// TwinCAT 3 PLC project Database_Code
// ProgramVersion: 3.1.4026.16
// libraries:
//   Tc2_Standard, * (Beckhoff Automation GmbH)
//   Tc2_System, * (Beckhoff Automation GmbH)
//   Tc2_Utilities, * (Beckhoff Automation GmbH)
//   Tc3_Database, * (Beckhoff Automation GmbH)
// project tree:
//   DUTs/ ST_SensorData.TcDUT
//   GVLs/ Global_Variables.TcGVL
//   / PlcTask.TcTTO
//   POUs/ CapacitiveConvert.TcPOU, FB_BufferManager.TcPOU, EncoderConvert.TcPOU, FC_SQL_InsertCommands_Capacitief.TcPOU, FC_SQL_InsertCommands_Encoder.TcPOU, FC_SQL_InsertCommands_TempSensor.TcPOU, FC_SQL_InsertCommands_LoadCell.TcPOU, LoadcellConvert.TcPOU, MAIN.TcPOU, TempConvert.TcPOU, TestCase.TcPOU
// real-time tasks:
//   TASK PlcTask: cycle T#5ms, priority 20, ADS port 350
// I/O:
//   DEVICE Device 3 (EtherCAT), AmsNetId 10.100.5.10.4.1
//     Term 6 (EK1100) [EK1100 EtherCAT Coupler (2A E-Bus)]
//       Term 7 (EL3074) [EL3074 4Ch. Ana. Input +/-10V, +/-20mA]
//       Term 8 (EL5032) [EL5032 2Ch. EnDat Encoder]
//       Term 9 (EL3204) [EL3204 4Ch. Ana. Input PT100 (RTD)]
//       Term 10 (EL7031) [EL7031 1Ch. Stepper motor output stage (24V, 1.5A)]
//       Term 12 (EL1819) [EL1819 16Ch. Dig. Input 24V, 10µs]
//       Term 13 (EL4004) [EL4004 4Ch. Ana. Output 0-10V, 12bit]
//       Term 16 (EL2809) [EL2809 16Ch. Dig. Output 24V, 0.5A]
//       Term 17 (EL9011) [EL9011 End Terminal]
// variable links:
//   Database_Code/Database_Code Instance <-> Device 3 (EtherCAT)/Term 6 (EK1100)/Term 10 (EL7031)
//     PlcTask Inputs/MAIN.RealMotorPosition <-> ENC Status/Counter value
//     PlcTask Inputs/MAIN.iLichtSluisValue1 <-> STM Status/Status/Digital input 1
//     PlcTask Inputs/MAIN.iLichtSluisValue2 <-> STM Status/Status/Digital input 2
//     PlcTask Inputs/MAIN.iMotorBusy <-> POS Status/Status/Busy
//     PlcTask Inputs/MAIN.iMotorCalibrated <-> POS Status/Status/Calibrated
//     PlcTask Inputs/MAIN.iMotorReady <-> POS Status/Status/Ready to execute
//     PlcTask Inputs/MAIN.iMotorStatus <-> POS Status/Status/Error
//     PlcTask Inputs/MAIN.iMotorWarning <-> POS Status/Status/Warning
//     PlcTask Outputs/MAIN.oEnableStart <-> ENC Control/Control/Set counter
//     PlcTask Outputs/MAIN.oMotorEnable <-> STM Control/Control/Enable
//     PlcTask Outputs/MAIN.oMotorExecute <-> POS Control/Control/Execute
//     PlcTask Outputs/MAIN.oMotorPosition <-> POS Control/Target position
//     PlcTask Outputs/MAIN.oMotorReset <-> STM Control/Control/Reset
//     PlcTask Outputs/MAIN.oMotorStartType <-> POS Control/Start type
//     PlcTask Outputs/MAIN.oMotorVelocity <-> POS Control/Velocity
//     PlcTask Outputs/MAIN.oStartPosition <-> ENC Control/Set counter value
//   Database_Code/Database_Code Instance <-> Device 3 (EtherCAT)/Term 6 (EK1100)/Term 12 (EL1819)
//     PlcTask Inputs/MAIN.iSwitchPULL <-> Channel 2/Input
//     PlcTask Inputs/MAIN.iSwitchPUSH <-> Channel 1/Input
//   Database_Code/Database_Code Instance <-> Device 3 (EtherCAT)/Term 6 (EK1100)/Term 13 (EL4004)
//     PlcTask Outputs/MAIN.oLoadcellPressure <-> AO Outputs Channel 1/Analog output
//   Database_Code/Database_Code Instance <-> Device 3 (EtherCAT)/Term 6 (EK1100)/Term 16 (EL2809)
//     PlcTask Outputs/MAIN.oLoadcellPull <-> Channel 2/Output
//     PlcTask Outputs/MAIN.oLoadcellPush <-> Channel 1/Output
//   Database_Code/Database_Code Instance <-> Device 3 (EtherCAT)/Term 6 (EK1100)/Term 7 (EL3074)
//     PlcTask Inputs/MAIN.iCapacitief1Value <-> AI Standard Channel 2/Value
//     PlcTask Inputs/MAIN.iCapacitief2Value <-> AI Standard Channel 3/Value
//     PlcTask Inputs/MAIN.iLoadCellValue <-> AI Standard Channel 1/Value
//   Database_Code/Database_Code Instance <-> Device 3 (EtherCAT)/Term 6 (EK1100)/Term 8 (EL5032)
//     PlcTask Inputs/MAIN.iEncoderValue <-> FB Inputs Channel 1 compact/Position
//   Database_Code/Database_Code Instance <-> Device 3 (EtherCAT)/Term 6 (EK1100)/Term 9 (EL3204)
//     PlcTask Inputs/MAIN.iTempSensor{1..4}Value <-> RTD Inputs Channel {1..4}/Value  (4 links)

CONFIGURATION Database_Code
    RESOURCE PLC ON TwinCAT3
        TASK PlcTask(INTERVAL := T#5ms, PRIORITY := 20);
        PROGRAM MAIN WITH PlcTask : MAIN;
    END_RESOURCE
END_CONFIGURATION

// ---- DUTs/ST_SensorData.TcDUT
TYPE ST_SensorData :
STRUCT
    SampleNumber    : INT;
    MeasurementNr   : INT;
    EncoderValue    : LREAL;
    Cap1Value       : LREAL;
    Cap2Value       : LREAL;
END_STRUCT
END_TYPE

// ---- GVLs/Global_Variables.TcGVL
VAR_GLOBAL
    g_aSensorBuffer : ARRAY[0..g_aSensorBuffers, 0..g_aSensorBufferSize] OF ST_SensorData; // aSensorBuffers buffers of aSensorBufferSize samples each
    g_aWriteSQL     : ARRAY[0..g_ASensorBuffers] OF BOOL;                 // Marks buffers ready for DB insert
	
END_VAR

VAR_GLOBAL CONSTANT
	g_aSensorBufferSize : INT := 999;
	g_aSensorBuffers : INT := 3600;
	sLocalID : STRING := '192.168.1.28.1.1'; //ams net id of database host
END_VAR

// ---- POUs/MAIN.TcPOU
PROGRAM MAIN
VAR CONSTANT
	//check variables
	PositiveDegrees : REAL := 0.1; 
	DifferenceDegrees : REAL := 0.1; 
	UpperBoundDegrees : INT := 9;
	LowerBoundDegrees : INT := -9;
	ZeroDegrees : REAL := 0.0;
	
	//convert variables
	ConvertToSec : INT := 1000;
	InvertDegrees : INT := -1;
	//time constant	
	tHomingStartInterval: TIME := T#25S;
	tHomingInterval: TIME := T#5S;
	tloadcellInterval: TIME := T#5S;
	//motor constants
	SlowestMotorSpeed : INT := 100;
	FastestMotorSpeed : INT := 1500;
	DefaultMotorSpeed : INT := 500;
	MotorLeftEdge : UDINT := 314000;
	MotorRightEdge : UDINT := 0;
	MotorStartValue : UDINT := 157000;
END_VAR


VAR
    //database variables
	FB_SQLDatabaseEvt : FB_SQLDatabaseEvt(sNetID := sLocalID, tTimeout := T#10S);
    FB_SQLCommandEvt  : FB_SQLCommandEvt(sNetID := sLocalID, tTimeout := T#10S);
    FB_SQLResultEvt   : FB_SQLResultEvt(sNetID := sLocalID, tTimeout := T#10S);
	SQL_Commands: ARRAY[1..10] OF STRING(500);
	DataBase_Connection: BOOL := FALSE;
   
	//inputs from sensor
    iLoadCellValue AT %I*: INT;
	iLoadCellPreviousValue : INT;
	iTempSensor1Value AT %I*: INT;
	iTempSensor2Value AT %I*: INT;
	iTempSensor3Value AT %I*: INT;
	iTempSensor4Value AT %I*: INT;
	iEncoderValue AT %I*: UDINT;
	iLichtSluisValue1 AT %I* : BOOL;
	iLichtSluisValue2 AT %I* : BOOL;
	iCapacitief1Value AT %I* : INT;
	iCapacitief2Value AT %I* : INT;

	//Strings to insert
	iSensorIDs : ARRAY[1..4] OF INT := [1,2,3,4];
	fbBufferManager: FB_BufferManager;
	//sample control
	SampleDone : BOOL; 
	SampleTrigger: BOOL;
	InsertingDone : BOOL;
	// INSERT state machine control
	TempInsert: INT ;
	
	//HMI Outputs
	iEncoderMotor : REAL;
	iLoadCellMotor : INT;
	iMotorSpeed : INT;
	iMetingen : INT;
	iTijd : INT;
	iTijdMeting : INT;
	iTijdSample : INT;
	
	//hmi display variables
	Temp1Value: STRING;  
	Temp2Value: STRING;
	Temp3Value: STRING;
	Temp4Value: STRING;
	
	//hmi variables
	bConfirm : BOOL;
	bStart : BOOL;
	bStop : BOOL := TRUE;
	Process_Status : BOOL; 
	bStartEnabled: BOOL;
	bDatalogView : BOOL;
	bActuatorView : BOOL;
	
	//measurement control
	TijdConvertUitwijking : TIME;
	TijdConvertMeting : TIME;
	TijdConvertSample: TIME;
	tUitwijkingTimer: TON; (* Timer to control wait time *) 
	tMetingTimer : TON; (* Timer to control measurement time*)
	tInsertTimer: TON; (* Timer to control insert intervals *)
	MeasurementsCompleted : INT;
	RealMotorPosition AT %I* : UDINT;
	MeasurementState: INT;
	Click : BOOL;
	Startup : BOOL;
	InitialDegrees : LREAL;
	
	//motor controls
	oMotorEnable AT %Q*: BOOL;
	oMotorExecute AT %Q*: BOOL;
	oMotorVelocity AT %Q*: INT;
	oMotorPosition AT %Q*: UDINT;
	oStartPosition AT %Q* : UDINT;
	oEnableStart AT %Q* : BOOL;
	oMotorStartType AT %Q* : INT;
	oMotorReset AT %Q* : BOOL;
	iMotorStatus AT %I* : BOOL;
	iMotorCalibrated AT %I* : BOOL;
	iMotorReady AT %I* : BOOL;
	iMotorBusy AT %I* : BOOL;
	iMotorWarning AT %I* : BOOL;
	//Homing controls
	HomingEdgeR : F_TRIG;
	HomingEdgeL : F_TRIG;
	Homing : INT := 0;
	HomingDone : BOOL;
	HomingDelayTimer: TON;
	HomingStartTimer : TON;

	//motor loadcell control
	oLoadcellPush AT %Q* : BOOL;
	oLoadcellPull AT %Q* : BOOL;
	oLoadcellPressure AT %Q* : INT;
	iSwitchPUSH AT %I* : BOOL;
	iSwitchPULL AT %I* : BOOL := TRUE;
	LoadcellDelayTimer: TON;
	//conversion variables
	TestForce : INT;
	iEncoderDegrees: LREAL;
	CapacitiveDistance1 : LREAL;
	CapacitiveDistance2 : LREAL;

	LoadInsert: INT;
END_VAR

VAR PERSISTENT
		iSampleNr: INT;
END_VAR

//conversion variables for measurement and hmi control
iEncoderDegrees := EncoderConvert(iEncoderValue); 
TestForce := LoadcellConvert(iLoadCellValue);
CapacitiveDistance1 := CapacitiveConvert(iCapacitief1Value);
CapacitiveDistance2 := CapacitiveConvert(iCapacitief2Value);
Temp1Value := TempConvert(iTempSensor1Value);
Temp2Value := Tempconvert(iTempSensor2Value);
Temp3Value := TempConvert(iTempSensor3Value);
Temp4Value := TempConvert(iTempSensor4Value);

//make connection to the database
IF NOT DataBase_Connection THEN
    FB_SQLDatabaseEvt.Connect(hDBID := 1);  // Attempt to connect

    // Wait until the connection is established
    IF FB_SQLDatabaseEvt.bConnected THEN
        FB_SQLDatabaseEvt.CreateCmd(pSQLCommand := ADR(FB_SQLCommandEvt));
        DataBase_Connection := TRUE;
    END_IF;

END_IF


//check status of motor and reset if necessary
IF iMotorStatus OR NOT iMotorCalibrated THEN
    oMotorReset := TRUE;
ELSE
    oMotorReset := FALSE;
END_IF

//execute homing process
IF NOT HomingDone THEN
// === Edge Detection (run every cycle) ===	
HomingEdgeR(CLK := iLichtSluisValue2); // Falling edge
HomingEdgeL(CLK := iLichtSluisValue1); // Falling edge

// === Homing State Machine ===
CASE Homing OF
0: // Initialization
    oStartPosition := MotorStartValue;
    oEnableStart := TRUE;
    oEnableStart := FALSE;
    oMotorEnable := TRUE;
    oMotorVelocity := DefaultMotorSpeed;
	HomingDelayTimer(PT := tHomingInterval);
	HomingStartTimer(PT := tHomingStartInterval);
    Homing := 1;

1: // Try moving CW
    IF iLichtSluisValue1 THEN
        oMotorPosition := MotorRightEdge;
        oMotorExecute := TRUE;
        Homing := 10;
    ELSE
        Homing := 2; // Try CCW
    END_IF

2: // Try moving CCW
    IF iLichtSluisValue2 THEN
        oMotorPosition := MotorLeftEdge;
        oMotorExecute := TRUE;
        Homing := 10;
    ELSE
        Homing := 1; // Back to CW
    END_IF

10: // Wait for sensor falling edge (center detected)
	HomingStartTimer(IN:= TRUE);
    IF (HomingEdgeL.Q OR HomingEdgeR.Q) OR HomingStartTimer.Q THEN
        oMotorExecute := FALSE;
        Homing := 11;
    END_IF

11: // Finalize homing
    oStartPosition := MotorStartValue;
    oEnableStart := TRUE;
	//wait for motor to turn off 
	HomingDelayTimer(IN:= TRUE);
    IF HomingDelayTimer.Q THEN
        HomingDone := TRUE;
		oMotorEnable := FALSE;
    	oMotorExecute := FALSE;
    END_IF
END_CASE
END_IF
	
//loadcell switch control
LoadcellDelayTimer(IN:= TRUE);
IF LoadcellDelayTimer.Q  AND NOT bStart THEN   
//move loadcell based on switch input
IF iSwitchPUSH THEN
	//push loadcell
	oLoadcellPull := FALSE;
	oLoadcellPush := TRUE;
	oLoadcellPressure := oLoadcellPressure + 3;
	IF oLoadcellPressure > 32700 THEN
	oLoadCellPressure := 32700;
	END_IF		
ELSIF iSwitchPULL THEN
	//pull loadcell
	oLoadcellPush := FALSE;
	oLoadcellPull := TRUE;
	oLoadcellPressure := 0;
	IF oLoadcellPressure < 0 THEN
	oLoadCellPressure := 0;
	END_IF
ELSIF NOT iSwitchPULL AND NOT iSwitchPUSH THEN
	oLoadcellPush := FALSE;
	oLoadcellPull := FALSE;	
END_IF
END_IF

	
//HMI Configuration
IF bConfirm AND HomingDone THEN
		TijdConvertUitwijking := INT_TO_TIME(iTijd) * ConvertToSec; //set to seconds
		TijdConvertMeting := INT_TO_TIME(iTijdMeting) * ConvertToSec; //set to seconds
		TijdConvertSample := INT_TO_TIME(iTijdSample) * ConvertToSec; //set to seconds
		IF iEncoderMotor > UpperBoundDegrees OR iEncoderMotor < LowerBoundDegrees THEN
		iEncoderMotor := ZeroDegrees;
		END_IF
		IF iMotorSpeed < SlowestMotorSpeed OR iMotorSpeed > FastestMotorSpeed THEN
			iMotorSpeed := DefaultMotorSpeed;
		END_IF
		bStartEnabled := TRUE;
		Startup := TRUE;
		//reset state for next measurement
		MeasurementState := 0;	
END_IF
//Measurement	
IF bStart AND HomingDone AND NOT bStop THEN

    CASE MeasurementState OF

      0: // Initialize
		//run this code only once
		IF Startup THEN	
        Process_Status := TRUE;
        oMotorEnable := TRUE;
        oMotorVelocity := iMotorSpeed;
        //Create timers
        tUitwijkingTimer(PT := TijdConvertUitwijking); 
        tMetingTimer(PT := TijdConvertMeting);
		tInsertTimer(PT := TijdConvertSample);
		oLoadcellPull := TRUE;
		oLoadCellPressure := 0;
		Startup := FALSE;
		END_IF
		
		IF TestForce < iLoadCellMotor THEN
			//push pnuematic
			oLoadcellPull := FALSE; 
			oLoadcellPush := TRUE;
			oLoadcellPressure := oLoadcellPressure + 3;
			IF oLoadcellPressure > 32700 THEN
			   oLoadCellPressure := 32700;
			END_IF		
		END_IF
		
		//loadcell is set at chosen Newtons 
        IF TestForce > iLoadCellMotor THEN
		//stop pnuematic
		oLoadcellPush := FALSE;
		oLoadcellPull := FALSE;	
		//Insert Loadcell value at Start 
		iSampleNr := iSampleNr + 1;
        //SQL_Commands[1] := FC_SQL_InsertCommands_LoadCell(LoadcellConvert(iLoadCellValue), iSampleNr, 0, MeasurementsCompleted);
        //FB_SQLCommandEvt.Execute(pSQLCmd := ADR(SQL_Commands[1]), cbSQLCmd := SIZEOF(SQL_Commands[1]));
		InitialDegrees := EncoderConvert(iEncoderValue);
		//go to next state
        MeasurementState := 1;
		END_IF

      1: //Wait at start
        tMetingTimer(IN := TRUE); // Start timer 
		  //wait before moving motor to chosen position			
        IF tMetingTimer.Q THEN 
		tInsertTimer(IN := TRUE); //start timer
		//insert data for buffer
		SampleTrigger := TRUE;
		SampleDone := FALSE; //stop Insert
		
		//insert temp sensor (and load sensor)
		SQL_Commands[1] := FC_SQL_InsertCommands_LoadCell(LoadcellConvert(iLoadCellValue), iSampleNr, 0, MeasurementsCompleted);
		SQL_Commands[3] := FC_SQL_InsertCommands_TempSensor(TempConvert(iTempSensor1Value), iSampleNr, iSensorIDs[1], MeasurementsCompleted);
		SQL_Commands[4] := FC_SQL_InsertCommands_TempSensor(TempConvert(iTempSensor2Value), iSampleNr, iSensorIDs[2], MeasurementsCompleted);
		SQL_Commands[7] := FC_SQL_InsertCommands_TempSensor(TempConvert(iTempSensor3Value), iSampleNr, iSensorIDs[3], MeasurementsCompleted);
		SQL_Commands[8] := FC_SQL_InsertCommands_TempSensor(TempConvert(iTempSensor4Value), iSampleNr, iSensorIDs[4], MeasurementsCompleted);
		CASE TempInsert OF
		0:	//execute Temp 1 INSERT
		IF FB_SQLCommandEvt.Execute(pSQLCmd := ADR(SQL_Commands[3]), cbSQLCmd := SIZEOF(SQL_Commands[3])) THEN
            TempInsert := 1;
        END_IF
		1:	//execute Temp 2 INSERT
		IF FB_SQLCommandEvt.Execute(pSQLCmd := ADR(SQL_Commands[4]), cbSQLCmd := SIZEOF(SQL_Commands[4])) THEN
            TempInsert := 2;
        END_IF
		2:	//execute Temp 3 INSERT
		IF FB_SQLCommandEvt.Execute(pSQLCmd := ADR(SQL_Commands[7]), cbSQLCmd := SIZEOF(SQL_Commands[7])) THEN
            TempInsert := 3;
        END_IF
		3:	//execute Temp 4 INSERT
		IF FB_SQLCommandEvt.Execute(pSQLCmd := ADR(SQL_Commands[8]), cbSQLCmd := SIZEOF(SQL_Commands[8])) THEN
            TempInsert := 4;
        END_IF
		4: //execute Load sensor insert
		IF FB_SQLCommandEvt.Execute(pSQLCmd := ADR(SQL_Commands[1]), cbSQLCmd := SIZEOF(SQL_Commands[1])) THEN
            TempInsert := 5;
        END_IF
		END_CASE
		
	
		
		 //sampling done move to position and insert data	
		 IF tInsertTimer.Q THEN
		 	SampleDone := TRUE; //start insert
			
            IF iEncoderMotor > PositiveDegrees THEN
                oMotorPosition := MotorLeftEdge; 
            ELSE
                oMotorPosition := MotorRightEdge;
            END_IF
			tInsertTimer(IN := FALSE); //stop timer
            oMotorExecute := TRUE;
            MeasurementState := 2;     
       	 END_IF
		END_IF
		
      2: //move to chosen degrees 
	    TempInsert := 0; //reset insert loop
        IF ABS(iEncoderDegrees - 	InitialDegrees) > ABS(iEncoderMotor)-  0.5 THEN
			oMotorVelocity := 100;
			IF ABS(iEncoderDegrees - 	InitialDegrees) > ABS(iEncoderMotor)- 0.25 THEN
				oMotorVelocity := 50;
				IF ABS(iEncoderDegrees - 	InitialDegrees)  > ABS(iEncoderMotor)  THEN
    	    	oMotorExecute := FALSE; //stop motor
            	tMetingTimer(IN := FALSE); // Stop Metingtimer
            	tUitwijkingTimer(IN := TRUE);  //start Uitijwkingtimer
				oMotorVelocity := iMotorSpeed;
				END_IF
			END_IF
        END_IF
        //wait at chosen degrees
        IF tUitwijkingTimer.Q THEN
            //Move motor back TO start position 
            oMotorPosition := oStartPosition;
            oMotorExecute := TRUE;
            MeasurementState := 3;     
        END_IF

      3: //restart measurement
        IF RealMotorPosition = oStartPosition THEN
            MeasurementsCompleted := MeasurementsCompleted + 1;
            tUitwijkingTimer(IN := FALSE); // Stop timer
            oMotorExecute := FALSE; //stop motor
			iEncoderMotor := iEncoderMotor * InvertDegrees;
            MeasurementState := 4;
        END_IF

      4: //check if measurments are complete
        IF MeasurementsCompleted = iMetingen THEN
            MeasurementsCompleted := 0;  
            MeasurementState := 5;
        ELSE
            MeasurementState := 1;     
        END_IF

      5: // Stop measurement
        bStop := TRUE; // reset bStop
        MeasurementState := 0; //reset state machine
		Click := TRUE;
    END_CASE
END_IF

// end measurements
IF bStop AND Click THEN
    Process_Status := FALSE; //hmi update
	bStart := FALSE;
	MeasurementState := 0; //reset state machine
	//reset loadcell
	oLoadcellPull := TRUE;
	oLoadCellPressure := 0;
	//insert done
	InsertingDone := fbBufferManager.bInsertingData;
	//home back to starter position
	IF(RealMotorPosition <> oStartPosition) THEN
		oMotorExecute := FALSE;
		oMotorPosition := oStartPosition;
		oMotorExecute := TRUE;
	ELSE
		oMotorEnable := FALSE;
    	oMotorExecute := FALSE;
		Click := FALSE;  
	END_IF	 
END_IF
	//insert buffer to database
	fbBufferManager(
    SampleDone := SampleDone,
	SampleTrigger := SampleTrigger,
    SampleNr := iSampleNr,
    MeasurementNr := MeasurementsCompleted,
    EncoderValue := iEncoderValue,
    Cap1Value := iCapacitief1Value,
    Cap2Value := iCapacitief2Value);

END_PROGRAM

// ---- POUs/FB_BufferManager.TcPOU
FUNCTION_BLOCK FB_BufferManager
VAR_INPUT
    SampleDone : BOOL;
	SampleTrigger : BOOL;
    SampleNr : INT;
    MeasurementNr : INT;
    EncoderValue : UDINT;
    Cap1Value : INT;
    Cap2Value : INT;
END_VAR
VAR
    // Buffer data
    nWriteIndex       : INT := 0;
    nWriteBufferIndex : INT := 0;
    nInsertIdx        : INT := 0;
    nSQLIndex         : INT := 0;
    InsertState       : INT := 0;
    InsertTriggered   : BOOL := FALSE;
    iSensorIDs : ARRAY[1..2] OF INT := [1,2];
	
    // SQL
    FB_SQLCommandEvt  : FB_SQLCommandEvt(sNetID := sLocalID, tTimeout := T#10S);
	FB_SQLDatabaseEvt : FB_SQLDatabaseEvt(sNetID := sLocalID, tTimeout := T#10S);
    SQL_Commands : ARRAY[1..10] OF STRING(500);
	DataBase_Connection: BOOL := FALSE;
	
	bAllInserted: BOOL;
	idx: INT;
END_VAR
VAR_OUTPUT
	bInsertingData: BOOL;
END_VAR

//make connection to the database
IF NOT DataBase_Connection THEN
    FB_SQLDatabaseEvt.Connect(hDBID := 1);  // Attempt to connect

    // Wait until the connection is established
    IF FB_SQLDatabaseEvt.bConnected THEN
        FB_SQLDatabaseEvt.CreateCmd(pSQLCommand := ADR(FB_SQLCommandEvt));
        DataBase_Connection := TRUE;
    END_IF;

END_IF


// Handle sampling trigger
IF  NOT SampleDone AND SampleTrigger  THEN
    g_aSensorBuffer[nWriteBufferIndex, nWriteIndex].SampleNumber  := SampleNr;
    g_aSensorBuffer[nWriteBufferIndex, nWriteIndex].MeasurementNr := MeasurementNr;
    g_aSensorBuffer[nWriteBufferIndex, nWriteIndex].EncoderValue  := EncoderConvert(EncoderValue);
    g_aSensorBuffer[nWriteBufferIndex, nWriteIndex].Cap1Value     := CapacitiveConvert(Cap1Value);
    g_aSensorBuffer[nWriteBufferIndex, nWriteIndex].Cap2Value     := CapacitiveConvert(Cap2Value);
	
    nWriteIndex := nWriteIndex + 1;
	
	
    IF nWriteIndex > g_aSensorBufferSize THEN
   		 	nWriteIndex := 0;
    		g_aWriteSQL[nWriteBufferIndex] := TRUE;

    		nWriteBufferIndex := nWriteBufferIndex + 1;
    		IF nWriteBufferIndex >= g_aSensorBuffers THEN
       		   nWriteBufferIndex := 0;
    		END_IF
		END_IF
		
END_IF

// Handle insertion if SampleDone
    IF g_aWriteSQL[nSQLIndex]  AND  SampleDone THEN
		bInsertingData := TRUE; // Set flag when starting insertion
        CASE InsertState OF
        0: // Insert encoder
            IF NOT InsertTriggered THEN
                SQL_Commands[2] := FC_SQL_InsertCommands_Encoder(
                    g_aSensorBuffer[nSQLIndex, nInsertIdx].EncoderValue,
                    g_aSensorBuffer[nSQLIndex, nInsertIdx].SampleNumber,
                    g_aSensorBuffer[nSQLIndex, nInsertIdx].MeasurementNr
                );
                InsertTriggered := FB_SQLCommandEvt.Execute(
                    pSQLCmd := ADR(SQL_Commands[2]),
                    cbSQLCmd := SIZEOF(SQL_Commands[2])
                );
            ELSIF NOT FB_SQLCommandEvt.bBusy THEN
                InsertState := 1;
                InsertTriggered := FALSE;
            END_IF

        1: // Insert Cap1
            IF NOT InsertTriggered THEN
                SQL_Commands[5] := FC_SQL_InsertCommands_Capacitief(
                    g_aSensorBuffer[nSQLIndex, nInsertIdx].Cap1Value,
                    g_aSensorBuffer[nSQLIndex, nInsertIdx].SampleNumber,
                    iSensorIDs[1],
                    g_aSensorBuffer[nSQLIndex, nInsertIdx].MeasurementNr
                );
                InsertTriggered := FB_SQLCommandEvt.Execute(
                    pSQLCmd := ADR(SQL_Commands[5]),
                    cbSQLCmd := SIZEOF(SQL_Commands[5])
                );
            ELSIF NOT FB_SQLCommandEvt.bBusy THEN
                InsertState := 2;
                InsertTriggered := FALSE;
            END_IF

        2: // Insert Cap2
            IF NOT InsertTriggered THEN
                SQL_Commands[6] := FC_SQL_InsertCommands_Capacitief(
                    g_aSensorBuffer[nSQLIndex, nInsertIdx].Cap2Value,
                    g_aSensorBuffer[nSQLIndex, nInsertIdx].SampleNumber,
                    iSensorIDs[2],
                    g_aSensorBuffer[nSQLIndex, nInsertIdx].MeasurementNr
                );
                InsertTriggered := FB_SQLCommandEvt.Execute(
                    pSQLCmd := ADR(SQL_Commands[6]),
                    cbSQLCmd := SIZEOF(SQL_Commands[6])
                );
            ELSIF NOT FB_SQLCommandEvt.bBusy THEN
                InsertState := 3;
                InsertTriggered := FALSE;
            END_IF
          
        3:
           IF NOT FB_SQLCommandEvt.bBusy THEN
                nInsertIdx := nInsertIdx + 1;
				
                IF nInsertIdx > g_aSensorBufferSize  THEN
                    nInsertIdx := 0;
                    g_aWriteSQL[nSQLIndex] := FALSE;
                    nSQLIndex := nSQLIndex + 1;
                    IF nSQLIndex > nWriteBufferIndex  THEN
                        nSQLIndex := 0;
						
                    END_IF
				
                END_IF

                InsertState := 0;
                InsertTriggered := FALSE;
            END_IF



        END_CASE
    END_IF
(* Check if any write flags are still set *)
bAllInserted := TRUE;
FOR idx := 0 TO g_aSensorBuffers - 1 DO
    IF g_aWriteSQL[idx] THEN
        bAllInserted := FALSE;
        EXIT;
    END_IF
END_FOR

(* If done inserting everything *)
IF bAllInserted AND NOT FB_SQLCommandEvt.bBusy THEN
    bInsertingData := FALSE;
	//IF SampleDone THEN
     //Clear buffers now if not already cleared
      // MEMSET(Destaddr := ADR(g_aSensorBuffer), n := SIZEOF(g_aSensorBuffer), FillByte := 0);
      // MEMSET(Destaddr := ADR(g_aWriteSQL), n := SIZEOF(g_aWriteSQL), FillByte := 0);
	//END_IF
END_IF

END_FUNCTION_BLOCK

// ---- POUs/EncoderConvert.TcPOU
FUNCTION EncoderConvert : LREAL
VAR_INPUT
	iEncoderValue : UDINT;
END_VAR
VAR
	//CONSTANTS
	ENCODER_OFFSET : UDINT := 1305092900;
	ENCODER_CONVERSION : UDINT := 1637500000*180;
END_VAR

//convert raw value to Degrees
EncoderConvert := DINT_TO_LREAL(UDINT_TO_DINT(iEncoderValue) - 1305092900) / 163750000.0 * 180.0 / PI;

END_FUNCTION

// ---- POUs/CapacitiveConvert.TcPOU
FUNCTION CapacitiveConvert : LREAL
VAR_INPUT
	  iRawValue     : INT;     // EL3074 raw value
END_VAR
VAR
  
    fVoltage      : LREAL;   // Converted voltage from raw value
    fScaleFactor  : LREAL := 100;   // µm per volt (from CPL190/290 calibration)
END_VAR

// Convert raw value to voltage
fVoltage := INT_TO_LREAL(iRawValue)/32767.0 * 10.0 ;

// Convert voltage to distance (µm)
CapacitiveConvert := fVoltage * fScaleFactor;

END_FUNCTION

// ---- POUs/FC_SQL_InsertCommands_Encoder.TcPOU
FUNCTION FC_SQL_InsertCommands_Encoder : STRING(255)
VAR_INPUT
    iSensorValue: LREAL;
    iSampleNr: INT;
	iMeasurementNr: INT;
END_VAR

FC_SQL_InsertCommands_Encoder := 'INSERT INTO [db_accessadmin].[Encoder] (SensorValue, SampleNr, Time, MeasurementNr) VALUES (';
FC_SQL_InsertCommands_Encoder := CONCAT(FC_SQL_InsertCommands_Encoder, LREAL_TO_STRING(iSensorValue));
FC_SQL_InsertCommands_Encoder := CONCAT(FC_SQL_InsertCommands_Encoder, ', ');
FC_SQL_InsertCommands_Encoder := CONCAT(FC_SQL_InsertCommands_Encoder, INT_TO_STRING(iSampleNr));
FC_SQL_InsertCommands_Encoder := CONCAT(FC_SQL_InsertCommands_Encoder, ', GETDATE() ');
FC_SQL_InsertCommands_Encoder := CONCAT(FC_SQL_InsertCommands_Encoder, ', ');
FC_SQL_InsertCommands_Encoder := CONCAT(FC_SQL_InsertCommands_Encoder, INT_TO_STRING(iMeasurementNr));
FC_SQL_InsertCommands_Encoder := CONCAT(FC_SQL_InsertCommands_Encoder, ');');

END_FUNCTION

// ---- POUs/FC_SQL_InsertCommands_Capacitief.TcPOU
FUNCTION FC_SQL_InsertCommands_Capacitief : STRING(255)
VAR_INPUT
    iSensorValue: lREAL;
    iSampleNr: INT;
	iSensorID: INT;
	iMeasurementNr: INT; 
END_VAR

FC_SQL_InsertCommands_Capacitief := 'INSERT INTO [db_accessadmin].[Capacitief] (SensorValue, SampleNr, Time, SensorID, MeasurementNr) VALUES (';
FC_SQL_InsertCommands_Capacitief := CONCAT(FC_SQL_InsertCommands_Capacitief, LREAL_TO_STRING(iSensorValue));
FC_SQL_InsertCommands_Capacitief := CONCAT(FC_SQL_InsertCommands_Capacitief, ', ');
FC_SQL_InsertCommands_Capacitief := CONCAT(FC_SQL_InsertCommands_Capacitief, INT_TO_STRING(iSampleNr));
FC_SQL_InsertCommands_Capacitief := CONCAT(FC_SQL_InsertCommands_Capacitief, ', GETDATE(), ');
FC_SQL_InsertCommands_Capacitief := CONCAT(FC_SQL_InsertCommands_Capacitief, INT_TO_STRING(iSensorID));
FC_SQL_InsertCommands_Capacitief := CONCAT(FC_SQL_InsertCommands_Capacitief, ', ');
FC_SQL_InsertCommands_Capacitief := CONCAT(FC_SQL_InsertCommands_Capacitief, INT_TO_STRING(iMeasurementNr));
FC_SQL_InsertCommands_Capacitief := CONCAT(FC_SQL_InsertCommands_Capacitief, ');');

END_FUNCTION

// ---- POUs/LoadcellConvert.TcPOU
FUNCTION LoadcellConvert : INT
VAR_INPUT
	LoadCellValue : INT;
END_VAR
VAR
	Voltage : REAL;
END_VAR

// Convert raw value to voltage
Voltage := INT_TO_REAL(LoadCellValue)/32767 * 10;
//convert voltage to Newtons(N) 
LoadCellConvert := REAL_TO_INT(Voltage * 980.7);

END_FUNCTION

// ---- POUs/TempConvert.TcPOU
FUNCTION TempConvert : STRING
VAR_INPUT
	iTempSensorValue : INT;
END_VAR
VAR
END_VAR

TempConvert := CONCAT(INT_TO_STRING(iTempSensorValue / 10), '.');   // Whole number part
TempConvert := CONCAT(TempConvert, INT_TO_STRING(ABS(iTempSensorValue MOD 10)));  // Decimal part

END_FUNCTION

// ---- POUs/FC_SQL_InsertCommands_LoadCell.TcPOU
FUNCTION FC_SQL_InsertCommands_LoadCell : STRING(255)
VAR_INPUT
    iSensorValue: INT;
    iSampleNr: INT;
	iSensorID: INT;
	iMeasurementNr: INT;
END_VAR

FC_SQL_InsertCommands_LoadCell := 'INSERT INTO [db_accessadmin].[LoadCell] (SensorValue, SampleNr, Time, SensorID, MeasurementNr) VALUES (';
FC_SQL_InsertCommands_LoadCell := CONCAT(FC_SQL_InsertCommands_LoadCell, INT_TO_STRING(iSensorValue));
FC_SQL_InsertCommands_LoadCell := CONCAT(FC_SQL_InsertCommands_LoadCell, ', ');
FC_SQL_InsertCommands_LoadCell := CONCAT(FC_SQL_InsertCommands_LoadCell, INT_TO_STRING(iSampleNr));
FC_SQL_InsertCommands_LoadCell := CONCAT(FC_SQL_InsertCommands_LoadCell, ', GETDATE(), ');
FC_SQL_InsertCommands_LoadCell := CONCAT(FC_SQL_InsertCommands_LoadCell, INT_TO_STRING(iSensorID));
FC_SQL_InsertCommands_LoadCell := CONCAT(FC_SQL_InsertCommands_LoadCell, ', ');
FC_SQL_InsertCommands_LoadCell := CONCAT(FC_SQL_InsertCommands_LoadCell, INT_TO_STRING(iMeasurementNr));
FC_SQL_InsertCommands_LoadCell := CONCAT(FC_SQL_InsertCommands_LoadCell, ');');

END_FUNCTION

// ---- POUs/FC_SQL_InsertCommands_TempSensor.TcPOU
FUNCTION FC_SQL_InsertCommands_TempSensor : STRING(255)
VAR_INPUT
    iSensorValue: STRING;
    iSampleNr: INT;
	iSensorID: INT;
	iMeasurementNr: INT;
END_VAR

FC_SQL_InsertCommands_TempSensor := 'INSERT INTO [db_accessadmin].[TempSensor] (SensorValue, SampleNr, Time, SensorID, MeasurementNr) VALUES (';
FC_SQL_InsertCommands_TempSensor := CONCAT(FC_SQL_InsertCommands_TempSensor, iSensorValue);
FC_SQL_InsertCommands_TempSensor := CONCAT(FC_SQL_InsertCommands_TempSensor, ', ');
FC_SQL_InsertCommands_TempSensor := CONCAT(FC_SQL_InsertCommands_TempSensor, INT_TO_STRING(iSampleNr));
FC_SQL_InsertCommands_TempSensor := CONCAT(FC_SQL_InsertCommands_TempSensor, ', GETDATE(), ');
FC_SQL_InsertCommands_TempSensor := CONCAT(FC_SQL_InsertCommands_TempSensor, INT_TO_STRING(iSensorID));
FC_SQL_InsertCommands_TempSensor := CONCAT(FC_SQL_InsertCommands_TempSensor, ', ');
FC_SQL_InsertCommands_TempSensor := CONCAT(FC_SQL_InsertCommands_TempSensor, INT_TO_STRING(iMeasurementNr));
FC_SQL_InsertCommands_TempSensor := CONCAT(FC_SQL_InsertCommands_TempSensor, ');');

END_FUNCTION

// ---- POUs/TestCase.TcPOU
FUNCTION TestCase : BOOL
VAR_INPUT
	
END_VAR
VAR
	//test case variables
 	CycleCounter : INT := 0;
    State : INT := 0;
	TargetPosition: UDINT;
	WaitingAtMid : BOOL;
	//timer for motor delay
	tHomeTimer: TON;
	tHomeInterval: TIME := T#10S;
	//variables that needs to be connected to motor
	oMotorVelocity : INT;
	oMotorPosition : UDINT;
	oMotorExecute : BOOL;
	oStartPosition : UDINT;
	oMotorEnable : BOOL;
	RealMotorPosition : UDINT;
	iMotorReady : BOOL;
	iMotorBusy : BOOL;
END_VAR

//THIS MOVES THE MACHINE TO THE OUTER 2 POINTS FOR A NUMBER OF TIMES
//Copy to main to test it 
// === Test Movement State Machine ===
CASE State OF

0: // Initialization
    oMotorVelocity := 400;
	tHomeTimer(PT := tHomeInterval);
    WaitingAtMid := FALSE;
    State := 1;

1: // Prepare move
    IF iMotorReady THEN
        oMotorPosition := TargetPosition;
        oMotorExecute := TRUE;
        State := 2;
    END_IF

2: // Wait for motion to midpoint or endpoint
    IF NOT WaitingAtMid AND ABS(RealMotorPosition - oStartPosition) < 100 THEN
        oMotorExecute := FALSE; // Stop motor at center
        WaitingAtMid := TRUE;
		oMotorEnable := FALSE; //mark edit stop motor
    END_IF

    IF WaitingAtMid THEN
        tHomeTimer(IN := TRUE);
        IF tHomeTimer.Q THEN
			
			oMotorEnable := TRUE; //mark edit stop motor
            // Start move to end after wait
            oMotorPosition := TargetPosition;
            oMotorExecute := TRUE;
            WaitingAtMid := FALSE;
            //TimerDone := TRUE; // Optional flag to track post-wait move
            tHomeTimer(IN := FALSE);
        END_IF
    ELSE
        tHomeTimer(IN := FALSE);
    END_IF

    // Wait for endpoint after resume
    IF  ABS(RealMotorPosition - TargetPosition) < 100 THEN
        oMotorExecute := FALSE; // Stop after reaching end
        //TimerDone := FALSE;
        State := 3;
    END_IF

3: // Toggle position and increment counter
    IF TargetPosition = 0 THEN
        TargetPosition := 314000;
    ELSE
        TargetPosition := 0;
    END_IF

    CycleCounter := CycleCounter + 1;

    IF CycleCounter >= 5 THEN
        State := 4;
    ELSE
        State := 1;
    END_IF

4: // Final stop
    IF iMotorReady THEN
	oMotorPosition := oStartPosition;
    oMotorExecute := TRUE;
	END_IF
    IF NOT iMotorBusy THEN
        oMotorExecute := FALSE;
    END_IF

END_CASE

END_FUNCTION
